// SIMATIC S7-200 SMART project (STEP 7-Micro/WIN SMART), CPU SR40

ORGANIZATION_BLOCK MAIN:OB1
TITLE=程序注释
BEGIN
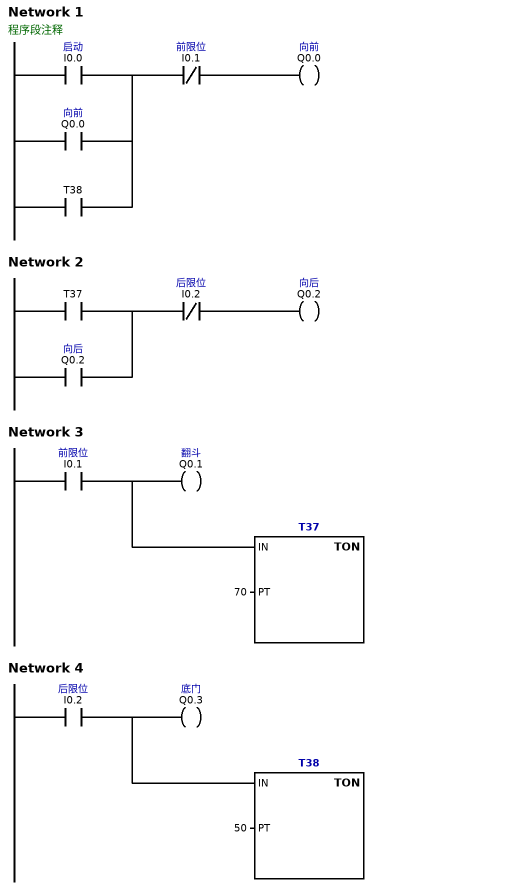
Network 1
// 程序段注释
LD     启动:I0.0
O      向前:Q0.0
O      T38
AN     前限位:I0.1
=      向前:Q0.0
Network 2
LD     T37
O      向后:Q0.2
AN     后限位:I0.2
=      向后:Q0.2
Network 3
LD     前限位:I0.1
=      翻斗:Q0.1
TON    T37, 70
Network 4
LD     后限位:I0.2
=      底门:Q0.3
TON    T38, 50
END_ORGANIZATION_BLOCK
